KUKA KRL program: test1.src

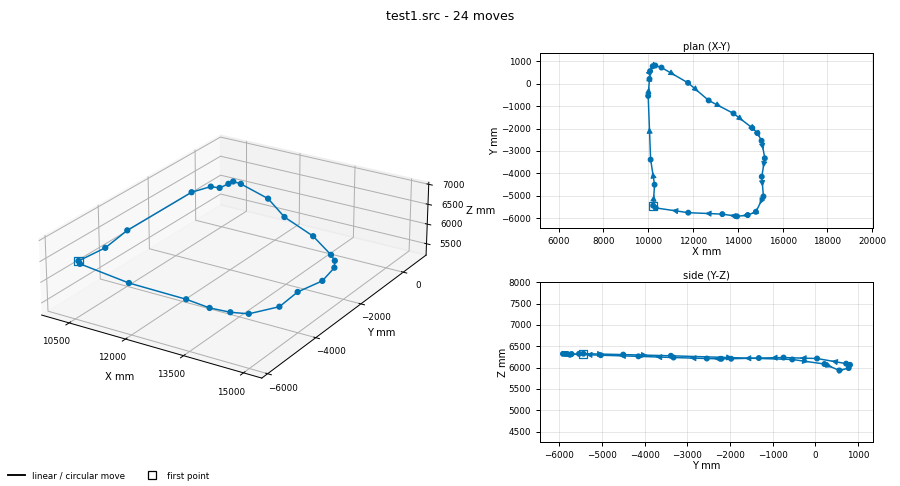
[picture p0: tool path of test1.src, 24 of 24 moves have a stored position in this frame; points joined in program order, loops and branches not executed]
&ACCESS RVP
&REL 1
&PARAM TEMPLATE_NAME = "LIN"
&PARAM EDITMASK = "KUKATP"
DEF KUKA_POINTS()
   ; X Y Z in mm, A B C in deg, Speed in mm/s
   $VEL.CP = 1 ; mm/s
   LIN {X 10219.431314, Y -5439.278844, Z 6326.879686, A -97.604650, B 9.465808, C -174.271067
   $VEL.CP = 130 ; mm/s
   LIN {X 10282.466366, Y -4504.990512, Z 6305.571894, A -105.939377, B 8.667205, C -175.121320
   $VEL.CP = 210 ; mm/s
   LIN {X 10106.555540, Y -3386.493702, Z 6277.723052, A -111.379282, B 7.935776, C -175.037403
   $VEL.CP = 212 ; mm/s
   LIN {X 9997.589816, Y -540.577204, Z 6191.201492, A -132.270569, B 10.107640, C 178.989263
   $VEL.CP = 157 ; mm/s
   LIN {X 10056.232742, Y 214.555058, Z 6084.481314, A -138.308058, B 10.518850, C 177.059371
   $VEL.CP = 128 ; mm/s
   LIN {X 10084.173688, Y 565.489142, Z 5933.643290, A -141.200936, B 12.114968, C 175.685238
   $VEL.CP = 106 ; mm/s
   LIN {X 10199.215556, Y 783.860906, Z 5989.464146, A -144.938819, B 12.573979, C 175.323929
   $VEL.CP = 96 ; mm/s
   LIN {X 10316.970514, Y 815.312260, Z 6065.961446, A -146.816539, B 12.771300, C 175.354666
   $VEL.CP = 133 ; mm/s
   LIN {X 10592.163278, Y 724.514482, Z 6093.622320, A -148.086106, B 10.177370, C 175.931309
   $VEL.CP = 170 ; mm/s
   LIN {X 11777.402552, Y 41.815580, Z 6213.573224, A -152.357779, B 8.362470, C 174.691477
   $VEL.CP = 63 ; mm/s
   LIN {X 12698.407134, Y -743.539140, Z 6236.018112, A -153.341433, B 7.177406, C 175.890865
   $VEL.CP = 177 ; mm/s
   LIN {X 13806.915400, Y -1324.061334, Z 6224.800916, A -150.852795, B 5.884993, C 174.251219
   $VEL.CP = 222 ; mm/s
   LIN {X 14646.224208, Y -1973.459704, Z 6208.190884, A -147.817673, B 3.628962, C 177.189584
   $VEL.CP = 217 ; mm/s
   LIN {X 14874.991254, Y -2203.470144, Z 6206.686002, A -145.974374, B 2.958120, C 177.719367
   $VEL.CP = 204 ; mm/s
   LIN {X 15059.237454, Y -2544.124418, Z 6213.417084, A -142.678380, B 3.076313, C 178.308006
   $VEL.CP = 181 ; mm/s
   LIN {X 15204.629936, Y -3325.230120, Z 6236.934892, A -136.732840, B 4.746079, C 179.974128
   $VEL.CP = 149 ; mm/s
   LIN {X 15068.174342, Y -4148.183638, Z 6264.463722, A -130.954265, B 4.558677, C -178.306176
   $VEL.CP = 120 ; mm/s
   LIN {X 15142.833182, Y -5030.695232, Z 6290.987832, A -125.060689, B 6.986184, C 179.890843
   $VEL.CP = 128 ; mm/s
   LIN {X 14807.377312, Y -5715.937142, Z 6318.827740, A -120.701391, B 7.219334, C -178.955236
   $VEL.CP = 141 ; mm/s
   LIN {X 14442.591888, Y -5860.824186, Z 6321.243766, A -119.275230, B 7.957412, C -178.141209
   $VEL.CP = 179 ; mm/s
   LIN {X 13962.795654, Y -5918.190786, Z 6323.398600, A -117.629531, B 9.433688, C -178.223764
   $VEL.CP = 222 ; mm/s
   LIN {X 13307.330338, Y -5818.567204, Z 6320.466438, A -117.811108, B 9.945480, C -177.489571
   $VEL.CP = 288 ; mm/s
   LIN {X 11786.877692, Y -5754.237622, Z 6301.139142, A -111.388571, B 11.565790, C -174.306411
   $VEL.CP = 47 ; mm/s
   LIN {X 10333.650210, Y -5541.719790, Z 6324.212310, A -95.179896, B 10.577539, C -170.878547
END
